SUBAPPLICATION Schneidwerk (* Subapplication Type *)
  (* Standard: 61499-2 *)
  (* Version 1.0, 2023-01-29, Franz *)
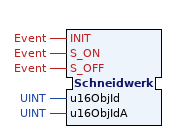
  EVENT_INPUT
    INIT;
    S_ON;
    S_OFF;
  END_EVENT
  VAR_INPUT
    u16ObjId : UINT;
    u16ObjIdA : UINT;
  END_VAR
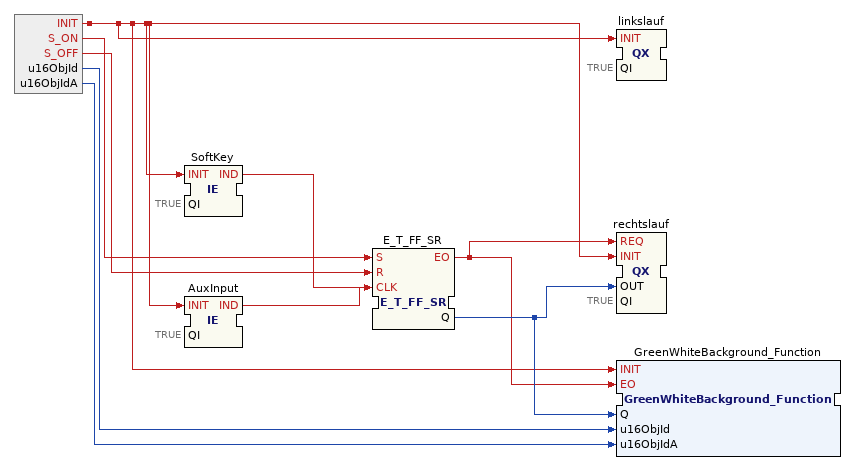
  (* TODO: Schneidwerk linkslauf bei jedem 2. Start. *)
  FBS
    rechtslauf : QX(QI := TRUE);
    E_T_FF_SR : E_T_FF_SR;
    linkslauf : QX(QI := TRUE);
    SoftKey : IE(QI := TRUE);
    AuxInput : IE(QI := TRUE);
  END_FBS
  SUBAPPS
    GreenWhiteBackground_Function : GreenWhiteBackground_Function;
  END_SUBAPPS
  EVENT_CONNECTIONS
    E_T_FF_SR.EO TO rechtslauf.REQ;
    S_ON TO E_T_FF_SR.S;
    S_OFF TO E_T_FF_SR.R;
    INIT TO linkslauf.INIT;
    INIT TO rechtslauf.INIT;
    INIT TO GreenWhiteBackground_Function.INIT;
    E_T_FF_SR.EO TO GreenWhiteBackground_Function.EO;
    INIT TO SoftKey.INIT;
    SoftKey.IND TO E_T_FF_SR.CLK;
    INIT TO AuxInput.INIT;
    AuxInput.IND TO E_T_FF_SR.CLK;
  END_CONNECTIONS
  DATA_CONNECTIONS
    E_T_FF_SR.Q TO rechtslauf.OUT;
    E_T_FF_SR.Q TO GreenWhiteBackground_Function.Q;
    u16ObjId TO GreenWhiteBackground_Function.u16ObjId;
    u16ObjIdA TO GreenWhiteBackground_Function.u16ObjIdA;
  END_CONNECTIONS
END_SUBAPPLICATION
